Staubli VAL3: setTool.pgx

program SetTool(tool x_tTool (dimensions=1), string x_sTool (dimensions=1))
begin
  $jogContext(x_tTool,world,0)
  if sLanguge=="Chinese"
    popUpMsg("切换当前工具已成"+x_sTool)
  else
    popUpMsg("Swtich the current tool to "+x_sTool)
  endIf
  tTool=x_tTool
  sTool=x_sTool
end
